Omron CX-Programmer project NewProject (CX-Programmer 9.75)

# PLC NewPLC1: CP2E-N N

## Global symbols (name address type ; comment)
Actuator_Mie D51 CHANNEL
0 CHANNEL  ; Pick Mie Kering 1
0.00 BOOL  ; Proxy Mie Kering 1
0.01 BOOL  ; PROXY BOWL DISPENSER
0.02 BOOL  ; START BUTTON
0.03 BOOL  ; Proxy Mie Kering 2
0.04 BOOL  ; Proxy Mie Kering 3
0.05 BOOL  ; Proxy Mie Kering 4
0.06 BOOL  ; Proxy Mie Kering 5
0.07 BOOL  ; Proxy Bowl Disp 1
0.08 BOOL  ; Proxy Bowl Disp 2
0.09 BOOL  ; Proxy Bowl Disp 3
1 CHANNEL  ; Pick Bowl 1
100.00 BOOL  ; MOTOR BOWL DISPENSER
100.01 BOOL  ; MOTOR KONVEYOR 1
100.02 BOOL  ; MOTOR KONVEYOR
100.06 BOOL  ; MOTOR LINEAR ACTUATOR 1
100.07 BOOL  ; MOTOR LINEAR ACTUATOR 2
101.00 BOOL  ; MOTOR LINEAR ACTUATOR 3
101.01 BOOL  ; MOTOR LINEAR ACTUATOR 4
101.02 BOOL  ; MOTOR LINEAR ACTUATOR 5
101.03 BOOL  ; Cup Disp 1
101.04 BOOL  ; Cup Disp 2
101.05 BOOL  ; Cup Disp 3
10.02 BOOL  ; Cup Dispensed
200.00 BOOL  ; RELAY START
200.01 BOOL  ; RELAY START KONVEYOR
200.02 BOOL  ; RELAY ACTUATOR
200.03 BOOL  ; MOTOR BOWL
200.04 BOOL  ; RESET COUNTER
C000 BOOL  ; Mie Kering Count
C001 BOOL  ; Cup Count
C003 BOOL  ; StockValidationMie
C004 BOOL  ; CupDisp Selector
C005 BOOL  ; StockValidationCup
C006 BOOL  ; DispensedCup_cnt
C007 BOOL  ; Dispensed Mie Kering
C008 BOOL  ; StockValidationMie
D130 CHANNEL  ; Boiling Time Mie 1
D131 CHANNEL  ; Time to pick Mie kering 2
D132 CHANNEL  ; Time to pick Mie kering 3
D133 CHANNEL  ; Boiling Time Mie 2
D134 CHANNEL  ; Boiling Time Mie 3
D30 CHANNEL  ; CupSelection
D31 CHANNEL  ; DispensedNoodle
D32 CHANNEL  ; NoodleSelector
D33 CHANNEL  ; Sisa Stock Mie
D34 CHANNEL  ; MinimumNoodle
D35 CHANNEL  ; Stock Cup
D36 CHANNEL  ; Sisa Cup Minimum
D5 CHANNEL  ; OrderQty (Local)
D6 CHANNEL  ; Order1_Menu (Local)
D7 CHANNEL  ; Order2_Menu (Local)
D8 CHANNEL  ; Order3_Menu (Local)
T000 BOOL  ; TIMER ActuatorMie
T001 BOOL  ; Cycle1 finish
T002 BOOL  ; Reset Second Cup
T003 BOOL  ; Rst Third Cup State
T004 BOOL  ; On MODBUS
T005 BOOL  ; TimerActuatorMie
T006 BOOL  ; Timer Boil Mie 1
T007 BOOL  ; Timer Pick Mie Kering 2
T008 BOOL  ; Timer Pick Mie Kering 3
T009 BOOL  ; Timer Boil Mie 2
T010 BOOL  ; Timer Boil Mie 3
T011 BOOL  ; Timer Actuator Mie 1
T012 BOOL  ; Timer Actuator Mie 2
T013 BOOL  ; Timer Actuator Mie 3
T014 BOOL  ; Timer Actuator Mie 4
T015 BOOL  ; Timer Actuator Mie 5
T016 BOOL  ; Timer CupDisp1
T017 BOOL  ; Timer CupDisp 3
T018 BOOL  ; Timer CupDisp3
W100.02 BOOL  ; Cup_Ready
W100.03 BOOL  ; Boiling_Mie1
W100.04 BOOL  ; Boiling_Mie2
W100.05 BOOL  ; Boiling_Mie3
W100.06 BOOL  ; RebusMie1_Done
W100.07 BOOL  ; RebusMie2_Done
W100.08 BOOL  ; RebusMie3_Done
W100.09 BOOL  ; Start_PickMie2_ToRobot
W100.10 BOOL  ; Start_PickMie3_ToRobot
W100.11 BOOL  ; Order1Topping
W100.12 BOOL  ; Order2Topping
W100.13 BOOL  ; Order3Topping
W101.00 BOOL  ; MieKering1_Ready
W101.01 BOOL  ; MieKering2_Ready
W101.02 BOOL  ; MieKering3_Ready
W101.03 BOOL  ; MieKering4_Ready
W101.04 BOOL  ; MieKering5_Ready
W102.00 BOOL  ; MieKering1 Picked
W102.01 BOOL  ; MieKering2 Picked
W102.02 BOOL  ; MieKering3 Picked
W102.03 BOOL  ; MieKering4 Picked
W102.04 BOOL  ; MieKering5 Picked
W102.05 BOOL  ; Cup1 Ready
W102.06 BOOL  ; Cup2 Ready
W102.07 BOOL  ; Cup3 Ready
W102.08 BOOL  ; Cup1 Picked
W102.09 BOOL  ; Cup2 Picked
W102.10 BOOL  ; Cup3 Picked
W10.00 BOOL  ; RST
W10.01 BOOL  ; MieKering_Picked
W10.02 BOOL  ; Cup dispensed
W10.03 BOOL  ; CupReady
W11.00 BOOL  ; Delay 1sec Trigger
W120.00 BOOL  ; Finished Order From Robot
W125.01 BOOL  ; Mie Kosong
W125.02 BOOL  ; Reset Stock
W125.03 BOOL  ; Set Timer
W125.04 BOOL  ; Cup Kosong
W12.00 BOOL  ; 1 Sec Delay
W1.00 BOOL  ; MieKering_Arrived
W1.01 BOOL  ; MieKering_Picked
W1.02 BOOL  ; Cup_Dropped
W2 CHANNEL  ; Multiple Order States
W20.00 BOOL  ; CheckOrder
W20.05 BOOL  ; Dispensing Done
W22.00 BOOL  ; On Mie
W22.01 BOOL  ; Inc_Cup
W22.02 BOOL  ; Inc_Mie
W2.00 BOOL  ; ModbusStatus
W2.01 BOOL  ; TIMRST
W2.02 BOOL  ; 1stOrder Done
W2.03 BOOL  ; Second Cup Done
W2.04 BOOL  ; All Cup Done
W2.05 BOOL  ; ThirdCup
W2.06 BOOL  ; Second Cup
W2.07 BOOL  ; Third Cup Done
W2.08 BOOL  ; LockActuatorMie
W3 CHANNEL  ; Object Position States
W30.00 BOOL  ; ProxyBowl1_Inverted
W30.01 BOOL  ; ProxyBowl2_Inverted
W30.02 BOOL  ; ProxyBowl3_Inverted
W30.03 BOOL  ; Cup3_State
W31.00 BOOL  ; Inv_ProxyMie1
W31.01 BOOL  ; Inv_ProxyMie2
W31.02 BOOL  ; Inv_ProxyMie3
W31.03 BOOL  ; Inv_ProxyMie4
W31.04 BOOL  ; Inv_ProxyMie5
W31.05 BOOL  ; Mie5_State
W31.06 BOOL  ; ResetMie5
W31.07 BOOL  ; ResetCup3
W3.00 BOOL  ; StartRelay
W3.01 BOOL  ; MotorMie
W3.02 BOOL  ; Conveyor
W3.03 BOOL  ; Mie Sampe
W3.04 BOOL  ; Set Sensor
W3.05 BOOL  ; BowlJatuh
W3.06 BOOL  ; Bowl Arrived
W3.07 BOOL  ; Second Cup
W4.00 BOOL  ; CupDisp Working
W5.00 BOOL  ; Start MODBUS
Cup1_Picked W21.03 BOOL
Cup2_Picked W21.04 BOOL
Cup3_Picked W21.05 BOOL
DispenserMieCnt C002 BOOL
FB_MODBUSTCP_SERVER _CP2E003_ExecuteModTcpServer
MieKering1_Picked W21.00 BOOL
MieKering2_Picked W21.01 BOOL
MieKering3_Picked W21.02 BOOL
Order1_Menu D110 CHANNEL  ; From PC
Order1_Topping1 D100 CHANNEL  ; From PC
Order1_Topping2 D101 CHANNEL  ; From PC
Order1_Topping3 D102 CHANNEL  ; From PC
Order2_Menu D111 CHANNEL  ; From PC
Order2_Topping1 D103 CHANNEL  ; From PC
Order2_Topping2 D104 CHANNEL  ; From PC
Order2_Topping3 D105 CHANNEL  ; From PC
Order3_Menu D112 CHANNEL  ; From PC
Order3_Topping1 D106 CHANNEL  ; From PC
Order3_Topping2 D107 CHANNEL  ; From PC
Order3_Topping3 D108 CHANNEL  ; From PC
Order_Quantity D120 CHANNEL  ; From PC
Start_Order W100.00 BOOL
StepNum D50 CHANNEL  ; Step Number

## Program CookingMie (cyclic task 0)
Local symbols
p_LT BOOL
p_eq BOOL
p_gt BOOL
p_lt BOOL

### Section MODBUS

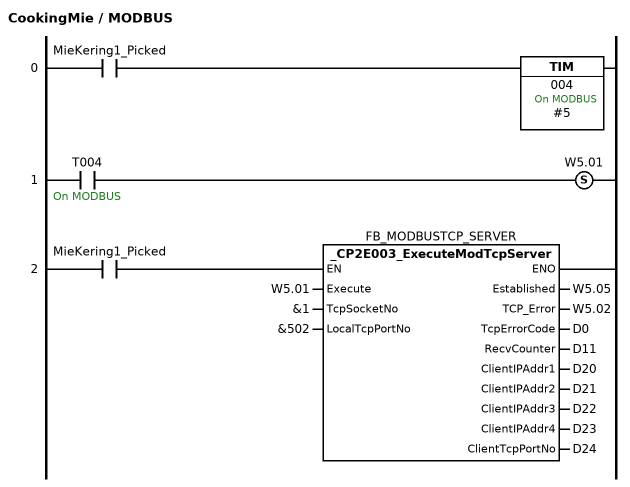
; rung 0
LD MieKering1_Picked
TIM 004 #5  ; On MODBUS
; rung 1
LD T004  ; On MODBUS
SET W5.01
; rung 2
LD MieKering1_Picked
CALL FB_MODBUSTCP_SERVER : _CP2E003_ExecuteModTcpServer (Execute := W5.01, TcpSocketNo := &1, LocalTcpPortNo := &502, Established => W5.05, TCP_Error => W5.02, TcpErrorCode => D0, RecvCounter => D11, ClientIPAddr1 => D20, ClientIPAddr2 => D21, ClientIPAddr3 => D22, ClientIPAddr4 => D23, ClientTcpPortNo => D24)

### Section Feeder_Main

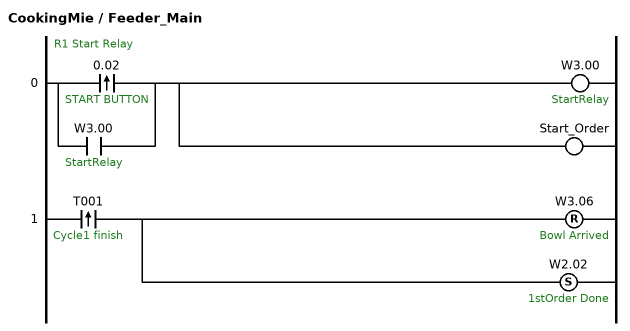
; rung 0: R1 Start Relay
@LD 0.02  ; START BUTTON
OR W3.00  ; StartRelay
OUT W3.00  ; StartRelay
OUT Start_Order
; rung 1
@LD T001  ; Cycle1 finish
RSET W3.06  ; Bowl Arrived
SET W2.02  ; 1stOrder Done

### Section Dispenser_Mie

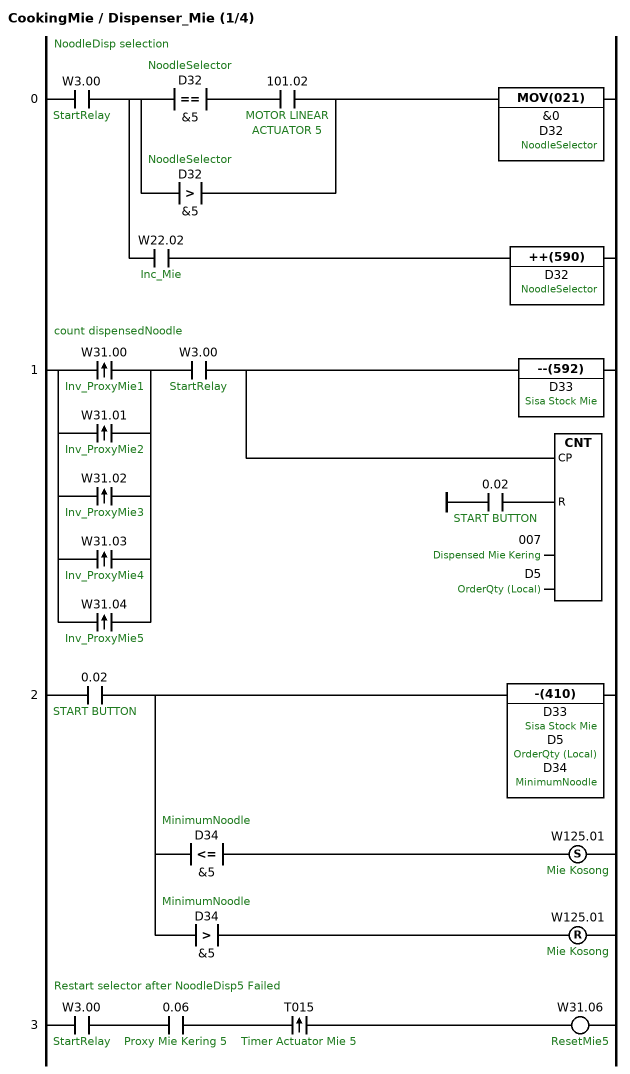
; rung 0: NoodleDisp selection
LD W3.00  ; StartRelay
OUT TR0
LD=(300) D32 &5  ; NoodleSelector
AND 101.02  ; MOTOR LINEAR ACTUATOR 5
OR>(320) D32 &5  ; NoodleSelector
ANDLD
MOV(021) &0 D32  ; NoodleSelector
LD TR0
AND W22.02  ; Inc_Mie
++(590) D32  ; NoodleSelector
; rung 1: count dispensedNoodle
@LD W31.00  ; Inv_ProxyMie1
@OR W31.01  ; Inv_ProxyMie2
@OR W31.02  ; Inv_ProxyMie3
@OR W31.03  ; Inv_ProxyMie4
@OR W31.04  ; Inv_ProxyMie5
AND W3.00  ; StartRelay
--(592) D33  ; Sisa Stock Mie
LD 0.02  ; START BUTTON
CNT 007 D5  ; OrderQty (Local), Dispensed Mie Kering
; rung 2
LD 0.02  ; START BUTTON
OUT TR0
-(410) D33 D5 D34  ; Sisa Stock Mie, OrderQty (Local), MinimumNoodle
AND<=(315) D34 &5  ; MinimumNoodle
SET W125.01  ; Mie Kosong
LD TR0
AND>(320) D34 &5  ; MinimumNoodle
RSET W125.01  ; Mie Kosong
; rung 3: Restart selector after NoodleDisp5 Failed
LD W3.00  ; StartRelay
AND 0.06  ; Proxy Mie Kering 5
@AND T015  ; Timer Actuator Mie 5
OUT W31.06  ; ResetMie5

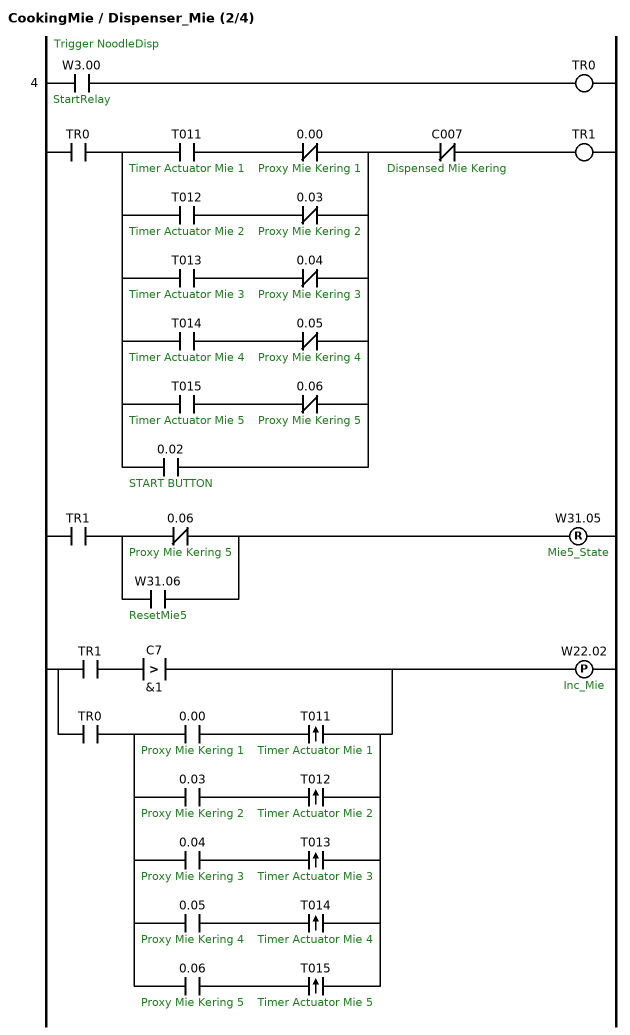
; rung 4: Trigger NoodleDisp
LD W3.00  ; StartRelay
OUT TR0
LD T011  ; Timer Actuator Mie 1
ANDNOT 0.00  ; Proxy Mie Kering 1
LD T012  ; Timer Actuator Mie 2
ANDNOT 0.03  ; Proxy Mie Kering 2
ORLD
LD T013  ; Timer Actuator Mie 3
ANDNOT 0.04  ; Proxy Mie Kering 3
ORLD
LD T014  ; Timer Actuator Mie 4
ANDNOT 0.05  ; Proxy Mie Kering 4
ORLD
LD T015  ; Timer Actuator Mie 5
ANDNOT 0.06  ; Proxy Mie Kering 5
ORLD
OR 0.02  ; START BUTTON
ANDLD
ANDNOT C007  ; Dispensed Mie Kering
OUT TR1
LDNOT 0.06  ; Proxy Mie Kering 5
OR W31.06  ; ResetMie5
ANDLD
RSET W31.05  ; Mie5_State
LD TR1
AND>(320) C7 &1
LD TR0
LD 0.00  ; Proxy Mie Kering 1
@AND T011  ; Timer Actuator Mie 1
LD 0.03  ; Proxy Mie Kering 2
@AND T012  ; Timer Actuator Mie 2
ORLD
LD 0.04  ; Proxy Mie Kering 3
@AND T013  ; Timer Actuator Mie 3
ORLD
LD 0.05  ; Proxy Mie Kering 4
@AND T014  ; Timer Actuator Mie 4
ORLD
LD 0.06  ; Proxy Mie Kering 5
@AND T015  ; Timer Actuator Mie 5
ORLD
ANDLD
ORLD
DIFU(013) W22.02  ; Inc_Mie

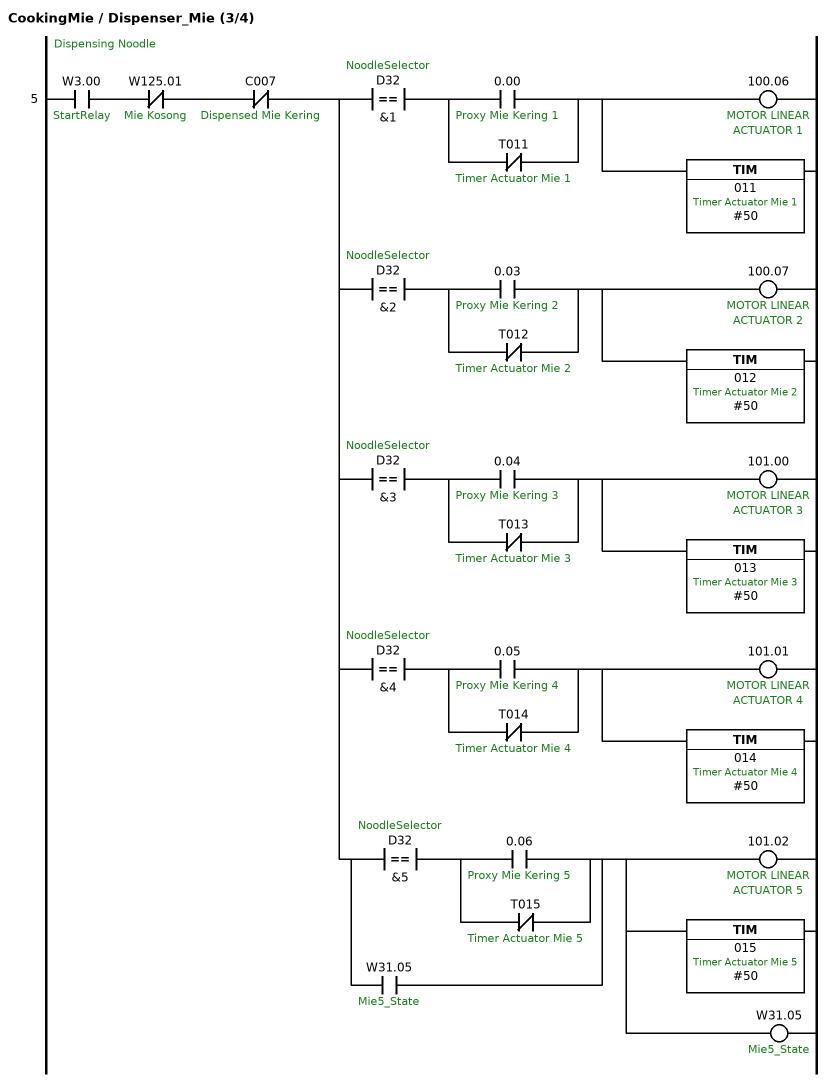
; rung 5: Dispensing Noodle
LD W3.00  ; StartRelay
ANDNOT W125.01  ; Mie Kosong
ANDNOT C007  ; Dispensed Mie Kering
OUT TR0
AND=(300) D32 &1  ; NoodleSelector
LD 0.00  ; Proxy Mie Kering 1
ORNOT T011  ; Timer Actuator Mie 1
ANDLD
OUT 100.06  ; MOTOR LINEAR ACTUATOR 1
TIM 011 #50  ; Timer Actuator Mie 1
LD TR0
AND=(300) D32 &2  ; NoodleSelector
LD 0.03  ; Proxy Mie Kering 2
ORNOT T012  ; Timer Actuator Mie 2
ANDLD
OUT 100.07  ; MOTOR LINEAR ACTUATOR 2
TIM 012 #50  ; Timer Actuator Mie 2
LD TR0
AND=(300) D32 &3  ; NoodleSelector
LD 0.04  ; Proxy Mie Kering 3
ORNOT T013  ; Timer Actuator Mie 3
ANDLD
OUT 101.00  ; MOTOR LINEAR ACTUATOR 3
TIM 013 #50  ; Timer Actuator Mie 3
LD TR0
AND=(300) D32 &4  ; NoodleSelector
LD 0.05  ; Proxy Mie Kering 4
ORNOT T014  ; Timer Actuator Mie 4
ANDLD
OUT 101.01  ; MOTOR LINEAR ACTUATOR 4
TIM 014 #50  ; Timer Actuator Mie 4
LD TR0
LD=(300) D32 &5  ; NoodleSelector
LD 0.06  ; Proxy Mie Kering 5
ORNOT T015  ; Timer Actuator Mie 5
ANDLD
OR W31.05  ; Mie5_State
ANDLD
OUT 101.02  ; MOTOR LINEAR ACTUATOR 5
TIM 015 #50  ; Timer Actuator Mie 5
OUT W31.05  ; Mie5_State

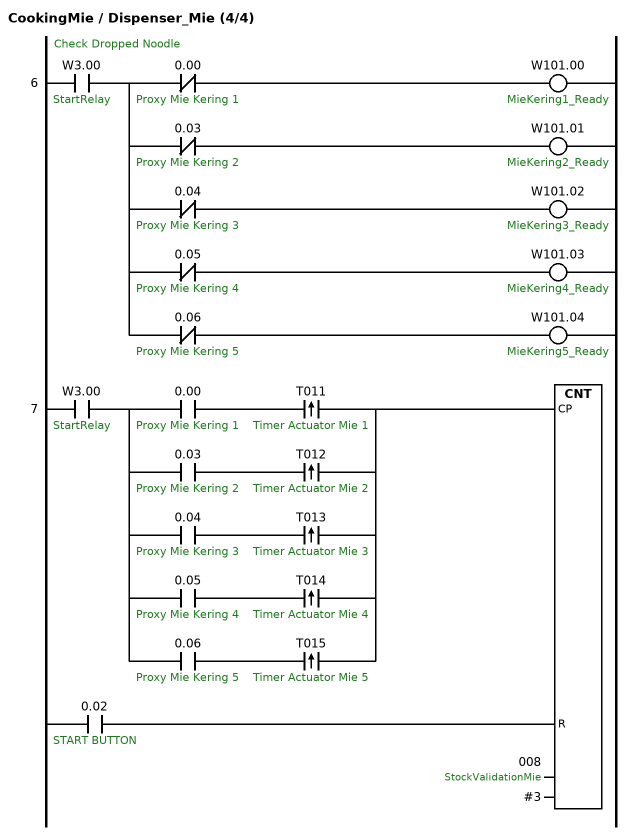
; rung 6: Check Dropped Noodle
LD W3.00  ; StartRelay
OUT TR0
ANDNOT 0.00  ; Proxy Mie Kering 1
OUT W101.00  ; MieKering1_Ready
LD TR0
ANDNOT 0.03  ; Proxy Mie Kering 2
OUT W101.01  ; MieKering2_Ready
LD TR0
ANDNOT 0.04  ; Proxy Mie Kering 3
OUT W101.02  ; MieKering3_Ready
LD TR0
ANDNOT 0.05  ; Proxy Mie Kering 4
OUT W101.03  ; MieKering4_Ready
LD TR0
ANDNOT 0.06  ; Proxy Mie Kering 5
OUT W101.04  ; MieKering5_Ready
; rung 7
LD W3.00  ; StartRelay
LD 0.00  ; Proxy Mie Kering 1
@AND T011  ; Timer Actuator Mie 1
LD 0.03  ; Proxy Mie Kering 2
@AND T012  ; Timer Actuator Mie 2
ORLD
LD 0.04  ; Proxy Mie Kering 3
@AND T013  ; Timer Actuator Mie 3
ORLD
LD 0.05  ; Proxy Mie Kering 4
@AND T014  ; Timer Actuator Mie 4
ORLD
LD 0.06  ; Proxy Mie Kering 5
@AND T015  ; Timer Actuator Mie 5
ORLD
ANDLD
LD 0.02  ; START BUTTON
CNT 008 #3  ; StockValidationMie

### Section Dispenser_Cup

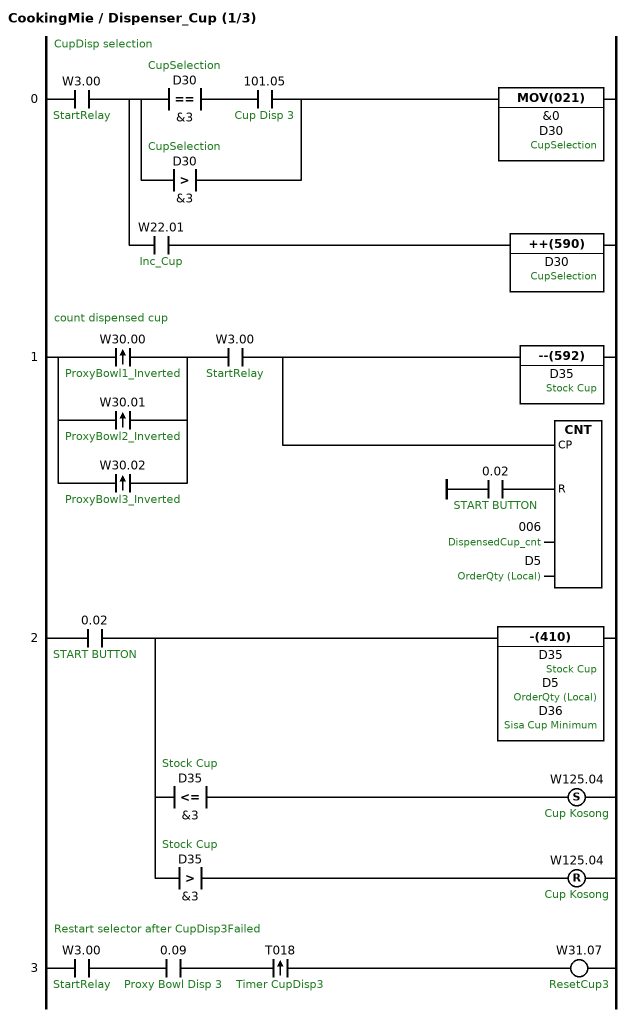
; rung 0: CupDisp selection
LD W3.00  ; StartRelay
OUT TR0
LD=(300) D30 &3  ; CupSelection
AND 101.05  ; Cup Disp 3
OR>(320) D30 &3  ; CupSelection
ANDLD
MOV(021) &0 D30  ; CupSelection
LD TR0
AND W22.01  ; Inc_Cup
++(590) D30  ; CupSelection
; rung 1: count dispensed cup
@LD W30.00  ; ProxyBowl1_Inverted
@OR W30.01  ; ProxyBowl2_Inverted
@OR W30.02  ; ProxyBowl3_Inverted
AND W3.00  ; StartRelay
--(592) D35  ; Stock Cup
LD 0.02  ; START BUTTON
CNT 006 D5  ; OrderQty (Local), DispensedCup_cnt
; rung 2
LD 0.02  ; START BUTTON
OUT TR0
-(410) D35 D5 D36  ; Stock Cup, OrderQty (Local), Sisa Cup Minimum
AND<=(315) D35 &3  ; Stock Cup
SET W125.04  ; Cup Kosong
LD TR0
AND>(320) D35 &3  ; Stock Cup
RSET W125.04  ; Cup Kosong
; rung 3: Restart selector after CupDisp3Failed
LD W3.00  ; StartRelay
AND 0.09  ; Proxy Bowl Disp 3
@AND T018  ; Timer CupDisp3
OUT W31.07  ; ResetCup3

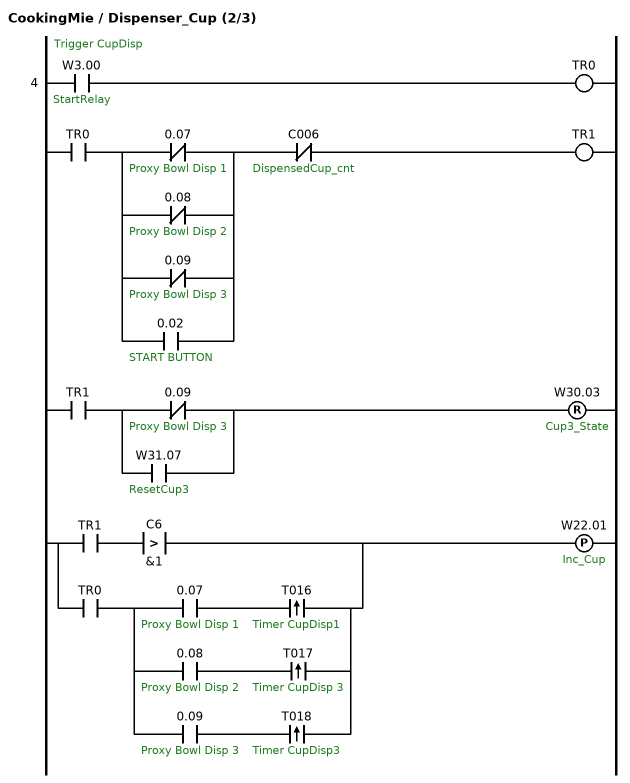
; rung 4: Trigger CupDisp
LD W3.00  ; StartRelay
OUT TR0
LDNOT 0.07  ; Proxy Bowl Disp 1
ORNOT 0.08  ; Proxy Bowl Disp 2
ORNOT 0.09  ; Proxy Bowl Disp 3
OR 0.02  ; START BUTTON
ANDLD
ANDNOT C006  ; DispensedCup_cnt
OUT TR1
LDNOT 0.09  ; Proxy Bowl Disp 3
OR W31.07  ; ResetCup3
ANDLD
RSET W30.03  ; Cup3_State
LD TR1
AND>(320) C6 &1
LD TR0
LD 0.07  ; Proxy Bowl Disp 1
@AND T016  ; Timer CupDisp1
LD 0.08  ; Proxy Bowl Disp 2
@AND T017  ; Timer CupDisp 3
ORLD
LD 0.09  ; Proxy Bowl Disp 3
@AND T018  ; Timer CupDisp3
ORLD
ANDLD
ORLD
DIFU(013) W22.01  ; Inc_Cup

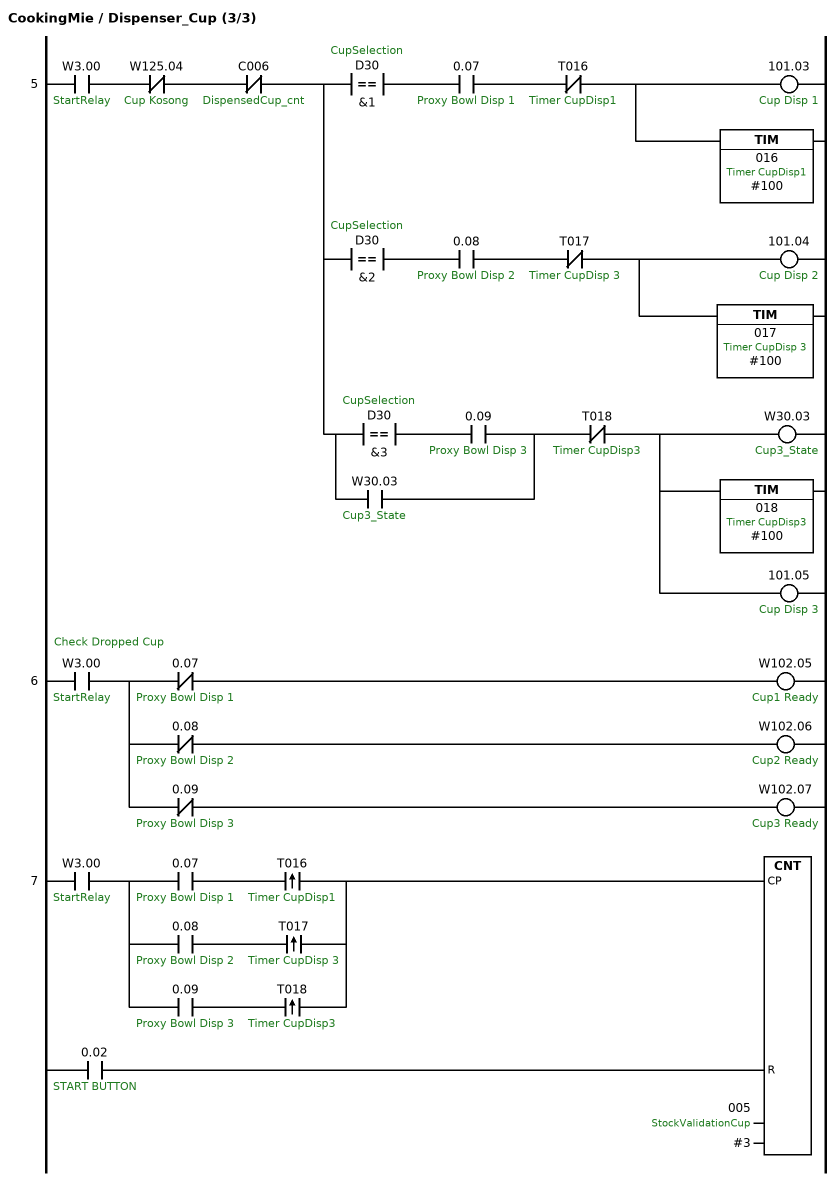
; rung 5
LD W3.00  ; StartRelay
ANDNOT W125.04  ; Cup Kosong
ANDNOT C006  ; DispensedCup_cnt
OUT TR0
AND=(300) D30 &1  ; CupSelection
AND 0.07  ; Proxy Bowl Disp 1
ANDNOT T016  ; Timer CupDisp1
OUT 101.03  ; Cup Disp 1
TIM 016 #100  ; Timer CupDisp1
LD TR0
AND=(300) D30 &2  ; CupSelection
AND 0.08  ; Proxy Bowl Disp 2
ANDNOT T017  ; Timer CupDisp 3
OUT 101.04  ; Cup Disp 2
TIM 017 #100  ; Timer CupDisp 3
LD TR0
LD=(300) D30 &3  ; CupSelection
AND 0.09  ; Proxy Bowl Disp 3
OR W30.03  ; Cup3_State
ANDLD
ANDNOT T018  ; Timer CupDisp3
OUT W30.03  ; Cup3_State
TIM 018 #100  ; Timer CupDisp3
OUT 101.05  ; Cup Disp 3
; rung 6: Check Dropped Cup
LD W3.00  ; StartRelay
OUT TR0
ANDNOT 0.07  ; Proxy Bowl Disp 1
OUT W102.05  ; Cup1 Ready
LD TR0
ANDNOT 0.08  ; Proxy Bowl Disp 2
OUT W102.06  ; Cup2 Ready
LD TR0
ANDNOT 0.09  ; Proxy Bowl Disp 3
OUT W102.07  ; Cup3 Ready
; rung 7
LD W3.00  ; StartRelay
LD 0.07  ; Proxy Bowl Disp 1
@AND T016  ; Timer CupDisp1
LD 0.08  ; Proxy Bowl Disp 2
@AND T017  ; Timer CupDisp 3
ORLD
LD 0.09  ; Proxy Bowl Disp 3
@AND T018  ; Timer CupDisp3
ORLD
ANDLD
LD 0.02  ; START BUTTON
CNT 005 #3  ; StockValidationCup

### Section Feeder_MultiOrder

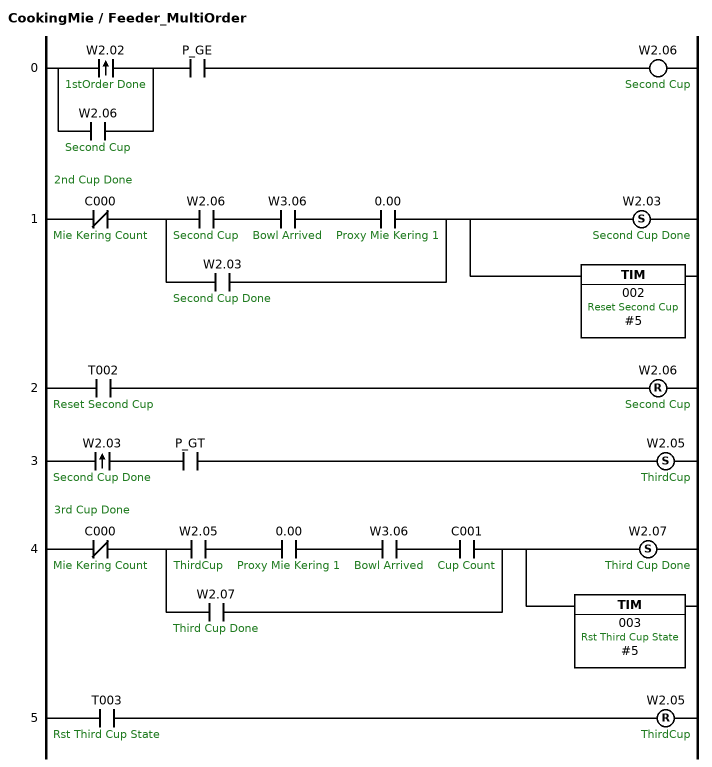
; rung 0
@LD W2.02  ; 1stOrder Done
OR W2.06  ; Second Cup
AND P_GE
OUT W2.06  ; Second Cup
; rung 1: 2nd Cup Done
LDNOT C000  ; Mie Kering Count
LD W2.06  ; Second Cup
AND W3.06  ; Bowl Arrived
AND 0.00  ; Proxy Mie Kering 1
OR W2.03  ; Second Cup Done
ANDLD
SET W2.03  ; Second Cup Done
TIM 002 #5  ; Reset Second Cup
; rung 2
LD T002  ; Reset Second Cup
RSET W2.06  ; Second Cup
; rung 3
@LD W2.03  ; Second Cup Done
AND P_GT
SET W2.05  ; ThirdCup
; rung 4: 3rd Cup Done
LDNOT C000  ; Mie Kering Count
LD W2.05  ; ThirdCup
AND 0.00  ; Proxy Mie Kering 1
AND W3.06  ; Bowl Arrived
AND C001  ; Cup Count
OR W2.07  ; Third Cup Done
ANDLD
SET W2.07  ; Third Cup Done
TIM 003 #5  ; Rst Third Cup State
; rung 5
LD T003  ; Rst Third Cup State
RSET W2.05  ; ThirdCup

### Section Cooking_Process

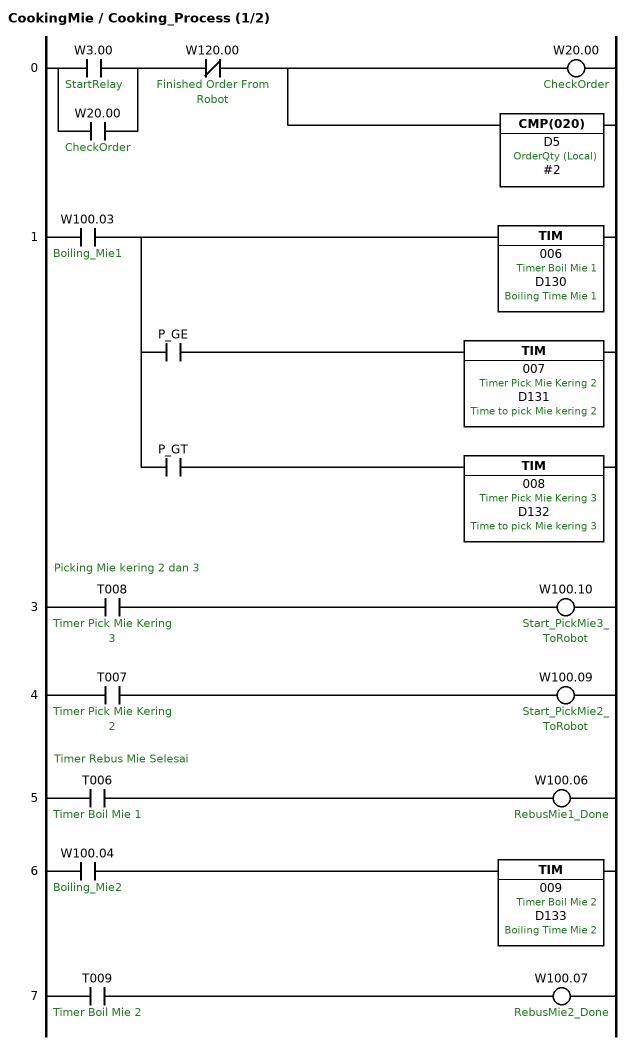
; rung 0
LD W3.00  ; StartRelay
OR W20.00  ; CheckOrder
ANDNOT W120.00  ; Finished Order From Robot
OUT W20.00  ; CheckOrder
CMP(020) D5 #2  ; OrderQty (Local)
; rung 1
LD W100.03  ; Boiling_Mie1
OUT TR0
TIM 006 D130  ; Boiling Time Mie 1, Timer Boil Mie 1
AND P_GE
TIM 007 D131  ; Time to pick Mie kering 2, Timer Pick Mie Kering 2
LD TR0
AND P_GT
TIM 008 D132  ; Time to pick Mie kering 3, Timer Pick Mie Kering 3
; rung 3: Picking Mie kering 2 dan 3
LD T008  ; Timer Pick Mie Kering 3
OUT W100.10  ; Start_PickMie3_ToRobot
; rung 4
LD T007  ; Timer Pick Mie Kering 2
OUT W100.09  ; Start_PickMie2_ToRobot
; rung 5: Timer Rebus Mie Selesai
LD T006  ; Timer Boil Mie 1
OUT W100.06  ; RebusMie1_Done
; rung 6
LD W100.04  ; Boiling_Mie2
TIM 009 D133  ; Boiling Time Mie 2, Timer Boil Mie 2
; rung 7
LD T009  ; Timer Boil Mie 2
OUT W100.07  ; RebusMie2_Done

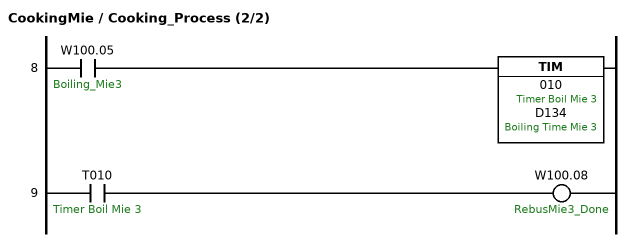
; rung 8
LD W100.05  ; Boiling_Mie3
TIM 010 D134  ; Boiling Time Mie 3, Timer Boil Mie 3
; rung 9
LD T010  ; Timer Boil Mie 3
OUT W100.08  ; RebusMie3_Done

### Section Order_Settings

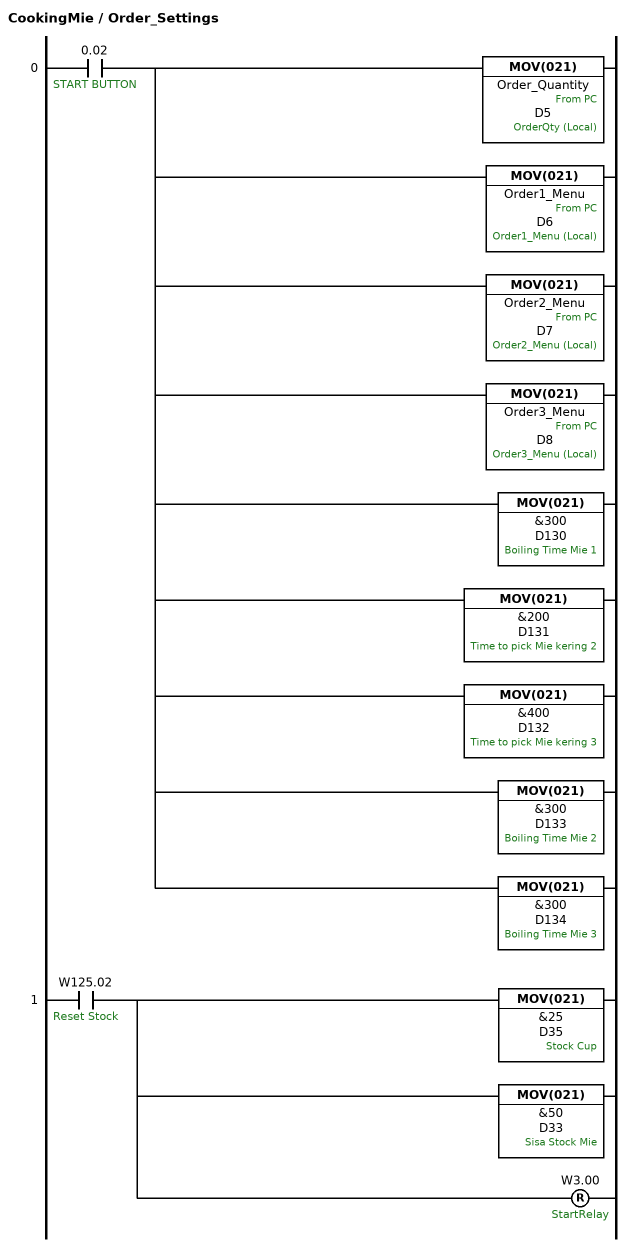
; rung 0
LD 0.02  ; START BUTTON
MOV(021) Order_Quantity D5  ; From PC, OrderQty (Local)
MOV(021) Order1_Menu D6  ; From PC, Order1_Menu (Local)
MOV(021) Order2_Menu D7  ; From PC, Order2_Menu (Local)
MOV(021) Order3_Menu D8  ; From PC, Order3_Menu (Local)
MOV(021) &300 D130  ; Boiling Time Mie 1
MOV(021) &200 D131  ; Time to pick Mie kering 2
MOV(021) &400 D132  ; Time to pick Mie kering 3
MOV(021) &300 D133  ; Boiling Time Mie 2
MOV(021) &300 D134  ; Boiling Time Mie 3
; rung 1
LD W125.02  ; Reset Stock
MOV(021) &25 D35  ; Stock Cup
MOV(021) &50 D33  ; Sisa Stock Mie
RSET W3.00  ; StartRelay

### Section RESET_States

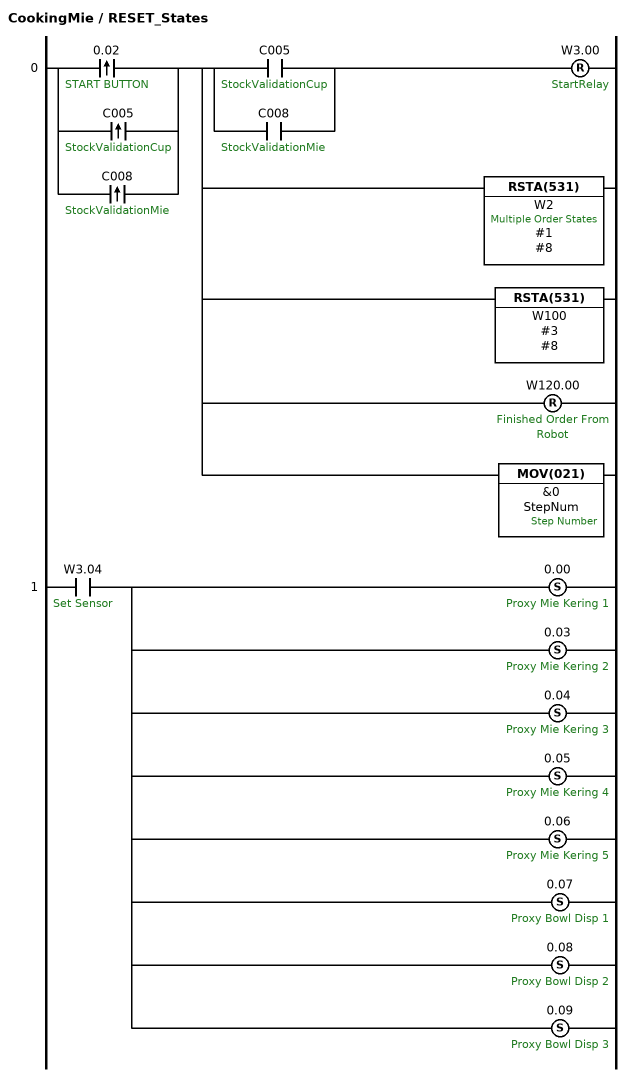
; rung 0
@LD 0.02  ; START BUTTON
@OR C005  ; StockValidationCup
@OR C008  ; StockValidationMie
OUT TR0
LD C005  ; StockValidationCup
OR C008  ; StockValidationMie
ANDLD
RSET W3.00  ; StartRelay
LD TR0
RSTA(531) W2 #1 #8  ; Multiple Order States
RSTA(531) W100 #3 #8
RSET W120.00  ; Finished Order From Robot
MOV(021) &0 StepNum  ; Step Number
; rung 1
LD W3.04  ; Set Sensor
SET 0.00  ; Proxy Mie Kering 1
SET 0.03  ; Proxy Mie Kering 2
SET 0.04  ; Proxy Mie Kering 3
SET 0.05  ; Proxy Mie Kering 4
SET 0.06  ; Proxy Mie Kering 5
SET 0.07  ; Proxy Bowl Disp 1
SET 0.08  ; Proxy Bowl Disp 2
SET 0.09  ; Proxy Bowl Disp 3

### Section Invert_Sensor

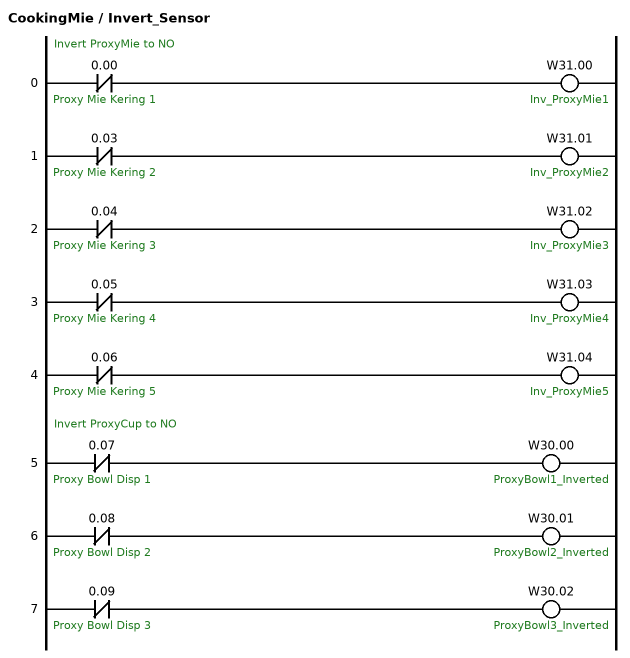
; rung 0: Invert ProxyMie to NO
LDNOT 0.00  ; Proxy Mie Kering 1
OUT W31.00  ; Inv_ProxyMie1
; rung 1
LDNOT 0.03  ; Proxy Mie Kering 2
OUT W31.01  ; Inv_ProxyMie2
; rung 2
LDNOT 0.04  ; Proxy Mie Kering 3
OUT W31.02  ; Inv_ProxyMie3
; rung 3
LDNOT 0.05  ; Proxy Mie Kering 4
OUT W31.03  ; Inv_ProxyMie4
; rung 4
LDNOT 0.06  ; Proxy Mie Kering 5
OUT W31.04  ; Inv_ProxyMie5
; rung 5: Invert ProxyCup to NO
LDNOT 0.07  ; Proxy Bowl Disp 1
OUT W30.00  ; ProxyBowl1_Inverted
; rung 6
LDNOT 0.08  ; Proxy Bowl Disp 2
OUT W30.01  ; ProxyBowl2_Inverted
; rung 7
LDNOT 0.09  ; Proxy Bowl Disp 3
OUT W30.02  ; ProxyBowl3_Inverted

### Section END
; rung 0
END(001)

## Function block _CP2E003_ExecuteModTcpServer (Omron library block, body left out)